///{attribute 'conditionalshow' := 'SomeText'}
///{attribute 'conditionalshow'}
///{attribute 'hide'}
VAR_GLOBAL
END_VAR

(* stored: Version 1.1.0.1, ProductVersion 3.1.4024.12
   GVL Constants: Id {61a71296-3b39-4b4c-9e67-cea520fcd5cc} *)
